FUNCTION_BLOCK E_REND_4 (* Like E_REND but with 4 inputs *)
  (* Standard: 61499-2 *)
  (* Version 1.0, 2017-06-07, Marc Jakobi, HTW Berlin *)
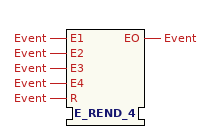
  EVENT_INPUT
    E1; (* First input event *)
    E2; (* Second input event *)
    E3; (* Third input event *)
    E4; (* Fourth input event *)
    R; (* Fith input event *)
  END_EVENT
  EVENT_OUTPUT
    EO; (* Output event *)
  END_EVENT
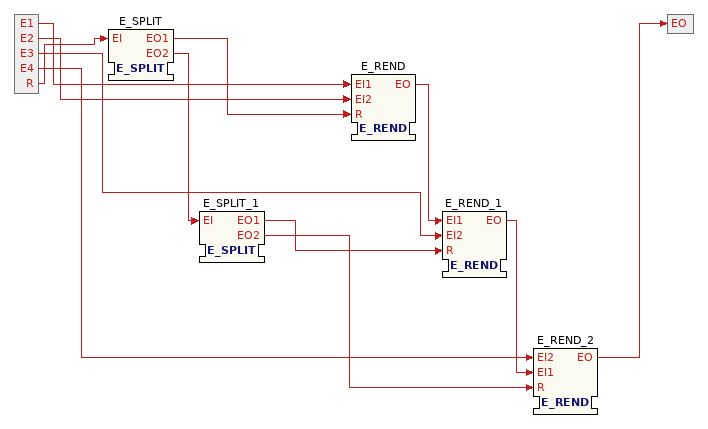
  FBS
    E_REND : E_REND;
    E_REND_1 : E_REND;
    E_REND_2 : E_REND;
    E_SPLIT : E_SPLIT;
    E_SPLIT_1 : E_SPLIT;
  END_FBS
  EVENT_CONNECTIONS
    E1 TO E_REND.EI1;
    E2 TO E_REND.EI2;
    E_REND.EO TO E_REND_1.EI1;
    E3 TO E_REND_1.EI2;
    E4 TO E_REND_2.EI2;
    E_REND_1.EO TO E_REND_2.EI1;
    R TO E_SPLIT.EI;
    E_SPLIT.EO1 TO E_REND.R;
    E_SPLIT.EO2 TO E_SPLIT_1.EI;
    E_SPLIT_1.EO1 TO E_REND_1.R;
    E_SPLIT_1.EO2 TO E_REND_2.R;
    E_REND_2.EO TO EO;
  END_CONNECTIONS
END_FUNCTION_BLOCK
